FUNCTION_BLOCK FB_MMA
VAR_OUTPUT
	iEtape:INT;
END_VAR
VAR
	fbEtape:FB_Etape;
	p_InitVar : p_InitVar;
END_VAR

fbEtape.mActualisation(FALSE,FALSE);

//activate ARU if system already running (fbEtape>10) and not in reset or already in ARU (fbEtape<800)
IF NOT fbBtn.xAru AND fbEtape.iNo>10 AND fbEtape.iNo<800 THEN
	fbEtape.piVal:=900; 
END_IF

//do reset
IF fbBtn.xReset AND fbEtape.iNo>10 AND fbEtape.iNo<800 THEN
	fbEtape.piVal:=800;
END_IF

CASE fbEtape.iNo OF
	0:fbEtape.psMess:='MMA | Booting MMA';
		fbEtape.piVal:=10;
	
	10:	fbEtape.psMess:='MMA | Init stock-Variables';
		//OB100 Siemens
		p_InitVar(); //initialiser les vars (propre a la machine)
		fbEtape.piVal:=50;
	
	50:fbEtape.psMess:='MMA | Selection du mode MMA';
		IF (stParam.stStatus.eMMA=Auto) THEN
			fbEtape.piVal:=300;
		ELSIF (stParam.stStatus.eMMA=Man) THEN
			fbEtape.piVal:=210;
		ELSIF (stParam.stStatus.eMMA=Init) THEN
			fbEtape.piVal:=100;
		END_IF
		
	//--------------------------------------------------------------
	//Init
	//--------------------------------------------------------------
	100:fbEtape.psMess:='MMA | Init | Wait for fbBtn.xStart';
		IF (fbBtn.xStart) THEN
			fbEtape.piVal:=110;
		ELSIF (stParam.stStatus.eMMA<>Init) THEN
			fbEtape.piVal:=50;
		END_IF
	110:fbEtape.psMess:='MMA | Init | Wait end';
		IF fbCycleInit.iEtape=999 THEN
		fbEtape.piVal:=50;
		END_IF
	111:fbEtape.psMess:='MMA | Init | Finished';
		IF fbCycleInit.xBusy THEN
		fbEtape.piVal:=50;
		END_IF
		
	//--------------------------------------------------------------
	//Manual
	//--------------------------------------------------------------
	210:fbEtape.psMess:='MMA | Manual | Wait for mode changing';
		IF (stParam.stStatus.eMMA<>Man) THEN
		fbEtape.piVal:=211;
		END_IF
	211:fbEtape.psMess:='MMA | Manual | Finishing';
		IF (fbCycleMan.xBusy) THEN
		fbEtape.piVal:=50;
		END_IF
		
	//--------------------------------------------------------------
	//Auto
	//--------------------------------------------------------------
	300:fbEtape.psMess:='MMA | Auto | Wait for fbBtn.xStart';
		IF fbBtn.xStart THEN
			fbEtape.piVal:=340;
		ELSIF (stParam.stStatus.eMMA<>Auto) THEN
			fbEtape.piVal:=50;
		END_IF
	
	340:fbEtape.psMess:='MMA | Auto | Do Init - Start';
		fbEtape.piVal:=341;
		
	341:fbEtape.psMess:='MMA | Auto | Do Init - Wait end';
		IF fbCycleInit.iEtape=999 THEN
			fbEtape.piVal:=350;
			stParam.stStatus.xInitOk:=TRUE;
		END_IF
		
	350:fbEtape.psMess:='MMA | Auto | Production - Wait Stop Signal';
		IF fbBtn.xStop THEN 
			fbEtape.piVal:=390;
		END_IF
		
	390:fbEtape.psMess:='MMA | Auto | Wait end';
		IF (NOT fbCycleAuto.xBusy) THEN
			fbEtape.piVal:=50;
		END_IF
		
	//--------------------------------------------------------------
	//Reset
	//--------------------------------------------------------------
	800:fbEtape.psMess:='MMA | Reset | Stopp all';
		fbEtape.piVal:=810;
	810:fbEtape.psMess:='MMA | Reset | Stopp all';
		fbEtape.piVal:=899;
	899:fbEtape.psMess:='MMA | Reset | Finished';
		IF fbBtn.xAirPressureOk THEN
			fbEtape.piVal:=50;
		END_IF
		
		
	//--------------------------------------------------------------
	//ARU
	//--------------------------------------------------------------
	900:fbEtape.psMess:='MMA | ARU | Stopp all';
		fbEtape.piVal:=910;
	910:fbEtape.psMess:='MMA | ARU | Stopp all';
		fbEtape.piVal:=950;
	950:fbEtape.psMess:='MMA | ARU | ok - Wait until resetting ARU-Btn';
		IF fbBtn.xAru THEN
			fbEtape.piVal:=999;
	END_IF
	999:fbEtape.psMess:='MMA | ARU | Finished';
		fbEtape.piVal:=50;
END_CASE

iEtape:=fbEtape.iNo;

END_FUNCTION_BLOCK

(* stored: Version 1.1.0.1, ProductVersion 3.1.4020.12
   POU FB_MMA: Id {0e7ce976-5b63-45cb-af38-a3b8fef59482}, SpecialFunc None *)
